PROGRAM prg_SearchString
VAR
	Persoon : Pers_data := (
		Name := 'Peeters',
		Firstname := 'Stijn',
		Address := 'Kerkstraat 12'
	);

	SearchFB : FB_SearchString;
	Result   : BOOL;
END_VAR

SearchFB(
	Person := Persoon,
	SearchTxt := 'stijn'
);

Result := SearchFB.Match;

END_PROGRAM

(* stored: Version 1.1.0.1, ProductVersion 3.1.4024.15
   POU prg_SearchString: Id {f413e5f4-2f33-48b8-97e6-0d917fead22f}, SpecialFunc None *)
